PROGRAM BasketToleranceCtrl
VAR
	ARfbStnToleranceCtrl		: ARRAY [0..iStnQty] OF fbToleranceTimeCtrl;

	tArm1ToleranceTimer		: TON;
	tArm1ToleranceTimerEV	: TIME;

	tArm2ToleranceTimer		: TON;
	tArm2ToleranceTimerEV	: TIME;

END_VAR

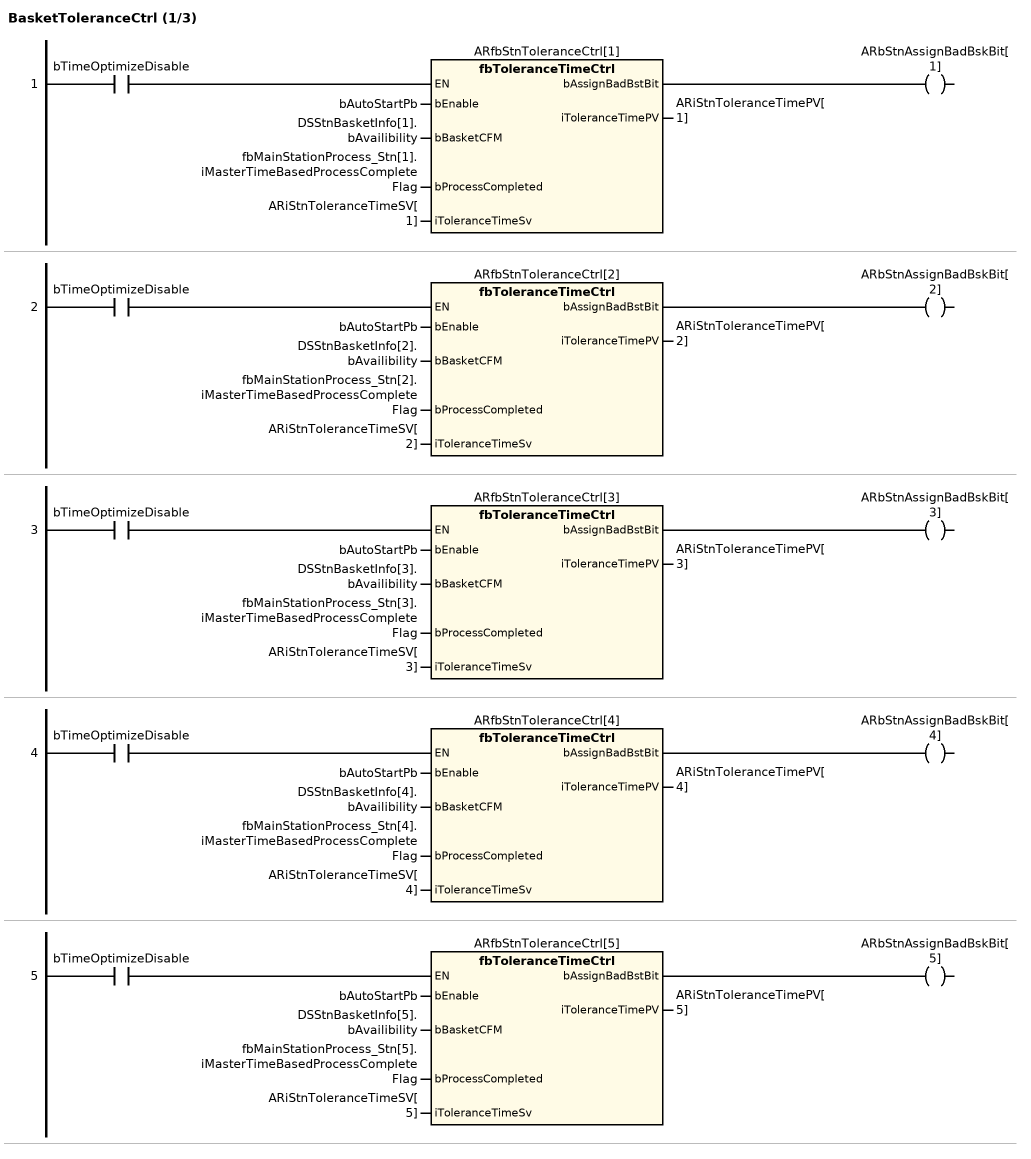
// NETWORK 1
IF bTimeOptimizeDisable THEN
    ARfbStnToleranceCtrl[1](
        bEnable := bAutoStartPb,
        bBasketCFM := DSStnBasketInfo[1].bAvailibility,
        bProcessCompleted := fbMainStationProcess_Stn[1].iMasterTimeBasedProcessCompleteFlag,
        iToleranceTimeSv := ARiStnToleranceTimeSV[1],
        iToleranceTimePV => ARiStnToleranceTimePV[1]); // fbToleranceTimeCtrl
END_IF
ARbStnAssignBadBskBit[1] := ARfbStnToleranceCtrl[1].bAssignBadBstBit;

// NETWORK 2
IF bTimeOptimizeDisable THEN
    ARfbStnToleranceCtrl[2](
        bEnable := bAutoStartPb,
        bBasketCFM := DSStnBasketInfo[2].bAvailibility,
        bProcessCompleted := fbMainStationProcess_Stn[2].iMasterTimeBasedProcessCompleteFlag,
        iToleranceTimeSv := ARiStnToleranceTimeSV[2],
        iToleranceTimePV => ARiStnToleranceTimePV[2]); // fbToleranceTimeCtrl
END_IF
ARbStnAssignBadBskBit[2] := ARfbStnToleranceCtrl[2].bAssignBadBstBit;

// NETWORK 3
IF bTimeOptimizeDisable THEN
    ARfbStnToleranceCtrl[3](
        bEnable := bAutoStartPb,
        bBasketCFM := DSStnBasketInfo[3].bAvailibility,
        bProcessCompleted := fbMainStationProcess_Stn[3].iMasterTimeBasedProcessCompleteFlag,
        iToleranceTimeSv := ARiStnToleranceTimeSV[3],
        iToleranceTimePV => ARiStnToleranceTimePV[3]); // fbToleranceTimeCtrl
END_IF
ARbStnAssignBadBskBit[3] := ARfbStnToleranceCtrl[3].bAssignBadBstBit;

// NETWORK 4
IF bTimeOptimizeDisable THEN
    ARfbStnToleranceCtrl[4](
        bEnable := bAutoStartPb,
        bBasketCFM := DSStnBasketInfo[4].bAvailibility,
        bProcessCompleted := fbMainStationProcess_Stn[4].iMasterTimeBasedProcessCompleteFlag,
        iToleranceTimeSv := ARiStnToleranceTimeSV[4],
        iToleranceTimePV => ARiStnToleranceTimePV[4]); // fbToleranceTimeCtrl
END_IF
ARbStnAssignBadBskBit[4] := ARfbStnToleranceCtrl[4].bAssignBadBstBit;

// NETWORK 5
IF bTimeOptimizeDisable THEN
    ARfbStnToleranceCtrl[5](
        bEnable := bAutoStartPb,
        bBasketCFM := DSStnBasketInfo[5].bAvailibility,
        bProcessCompleted := fbMainStationProcess_Stn[5].iMasterTimeBasedProcessCompleteFlag,
        iToleranceTimeSv := ARiStnToleranceTimeSV[5],
        iToleranceTimePV => ARiStnToleranceTimePV[5]); // fbToleranceTimeCtrl
END_IF
ARbStnAssignBadBskBit[5] := ARfbStnToleranceCtrl[5].bAssignBadBstBit;

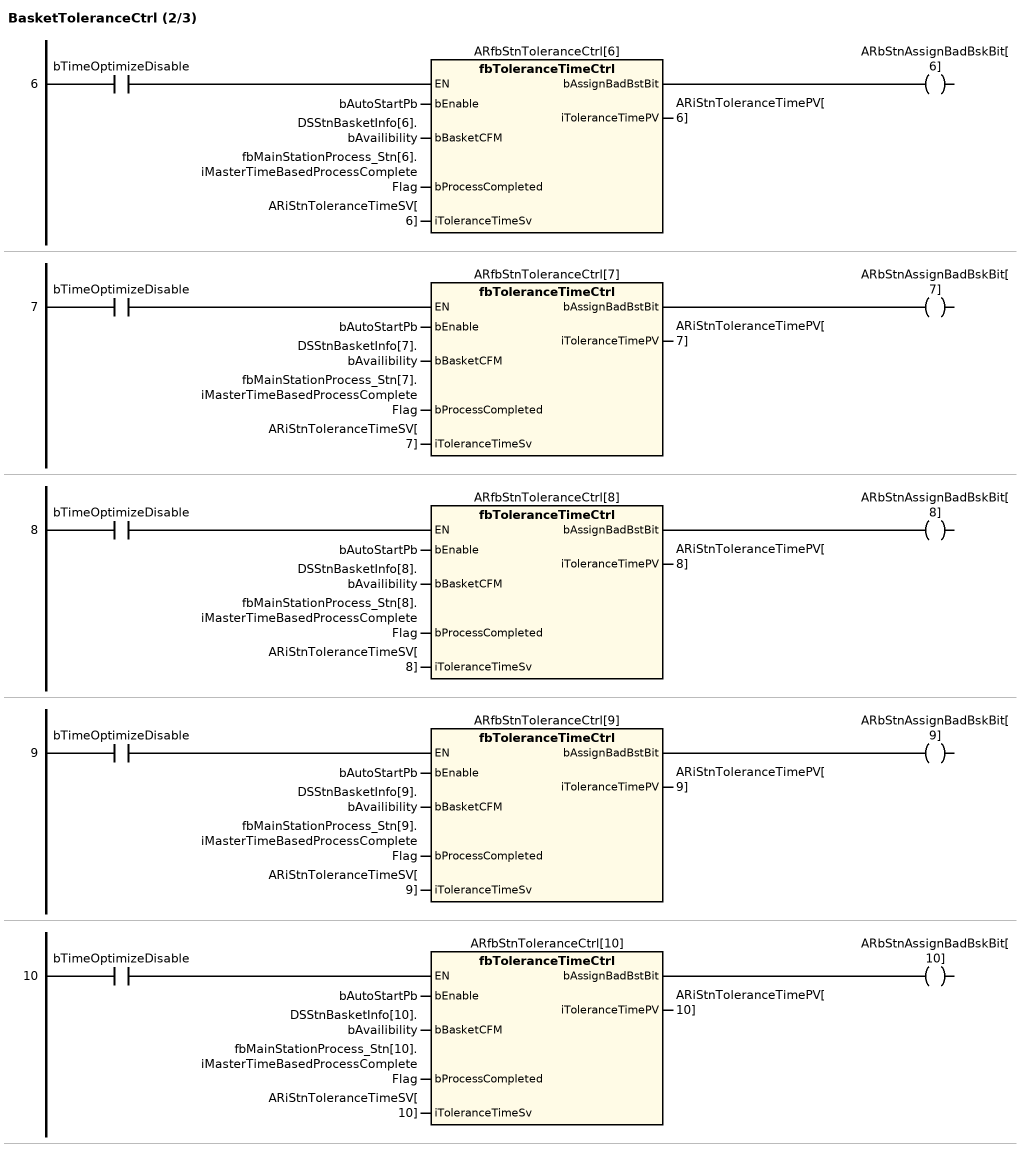
// NETWORK 6
IF bTimeOptimizeDisable THEN
    ARfbStnToleranceCtrl[6](
        bEnable := bAutoStartPb,
        bBasketCFM := DSStnBasketInfo[6].bAvailibility,
        bProcessCompleted := fbMainStationProcess_Stn[6].iMasterTimeBasedProcessCompleteFlag,
        iToleranceTimeSv := ARiStnToleranceTimeSV[6],
        iToleranceTimePV => ARiStnToleranceTimePV[6]); // fbToleranceTimeCtrl
END_IF
ARbStnAssignBadBskBit[6] := ARfbStnToleranceCtrl[6].bAssignBadBstBit;

// NETWORK 7
IF bTimeOptimizeDisable THEN
    ARfbStnToleranceCtrl[7](
        bEnable := bAutoStartPb,
        bBasketCFM := DSStnBasketInfo[7].bAvailibility,
        bProcessCompleted := fbMainStationProcess_Stn[7].iMasterTimeBasedProcessCompleteFlag,
        iToleranceTimeSv := ARiStnToleranceTimeSV[7],
        iToleranceTimePV => ARiStnToleranceTimePV[7]); // fbToleranceTimeCtrl
END_IF
ARbStnAssignBadBskBit[7] := ARfbStnToleranceCtrl[7].bAssignBadBstBit;

// NETWORK 8
IF bTimeOptimizeDisable THEN
    ARfbStnToleranceCtrl[8](
        bEnable := bAutoStartPb,
        bBasketCFM := DSStnBasketInfo[8].bAvailibility,
        bProcessCompleted := fbMainStationProcess_Stn[8].iMasterTimeBasedProcessCompleteFlag,
        iToleranceTimeSv := ARiStnToleranceTimeSV[8],
        iToleranceTimePV => ARiStnToleranceTimePV[8]); // fbToleranceTimeCtrl
END_IF
ARbStnAssignBadBskBit[8] := ARfbStnToleranceCtrl[8].bAssignBadBstBit;

// NETWORK 9
IF bTimeOptimizeDisable THEN
    ARfbStnToleranceCtrl[9](
        bEnable := bAutoStartPb,
        bBasketCFM := DSStnBasketInfo[9].bAvailibility,
        bProcessCompleted := fbMainStationProcess_Stn[9].iMasterTimeBasedProcessCompleteFlag,
        iToleranceTimeSv := ARiStnToleranceTimeSV[9],
        iToleranceTimePV => ARiStnToleranceTimePV[9]); // fbToleranceTimeCtrl
END_IF
ARbStnAssignBadBskBit[9] := ARfbStnToleranceCtrl[9].bAssignBadBstBit;

// NETWORK 10
IF bTimeOptimizeDisable THEN
    ARfbStnToleranceCtrl[10](
        bEnable := bAutoStartPb,
        bBasketCFM := DSStnBasketInfo[10].bAvailibility,
        bProcessCompleted := fbMainStationProcess_Stn[10].iMasterTimeBasedProcessCompleteFlag,
        iToleranceTimeSv := ARiStnToleranceTimeSV[10],
        iToleranceTimePV => ARiStnToleranceTimePV[10]); // fbToleranceTimeCtrl
END_IF
ARbStnAssignBadBskBit[10] := ARfbStnToleranceCtrl[10].bAssignBadBstBit;

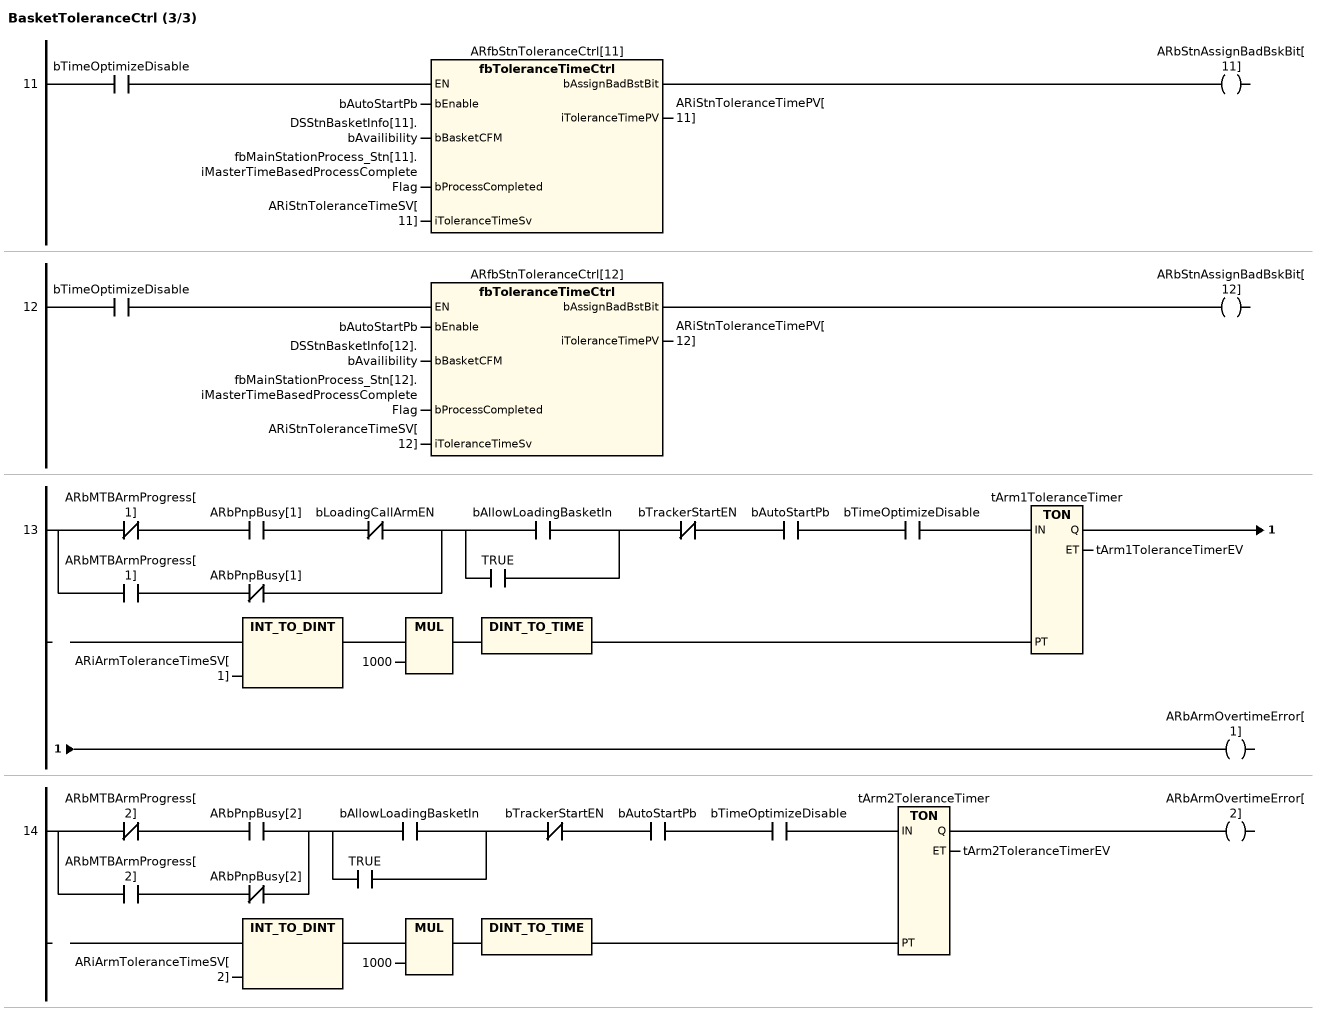
// NETWORK 11
IF bTimeOptimizeDisable THEN
    ARfbStnToleranceCtrl[11](
        bEnable := bAutoStartPb,
        bBasketCFM := DSStnBasketInfo[11].bAvailibility,
        bProcessCompleted := fbMainStationProcess_Stn[11].iMasterTimeBasedProcessCompleteFlag,
        iToleranceTimeSv := ARiStnToleranceTimeSV[11],
        iToleranceTimePV => ARiStnToleranceTimePV[11]); // fbToleranceTimeCtrl
END_IF
ARbStnAssignBadBskBit[11] := ARfbStnToleranceCtrl[11].bAssignBadBstBit;

// NETWORK 12
IF bTimeOptimizeDisable THEN
    ARfbStnToleranceCtrl[12](
        bEnable := bAutoStartPb,
        bBasketCFM := DSStnBasketInfo[12].bAvailibility,
        bProcessCompleted := fbMainStationProcess_Stn[12].iMasterTimeBasedProcessCompleteFlag,
        iToleranceTimeSv := ARiStnToleranceTimeSV[12],
        iToleranceTimePV => ARiStnToleranceTimePV[12]); // fbToleranceTimeCtrl
END_IF
ARbStnAssignBadBskBit[12] := ARfbStnToleranceCtrl[12].bAssignBadBstBit;

// NETWORK 13
tArm1ToleranceTimer(
    IN := ((NOT ARbMTBArmProgress[1] AND ARbPnpBusy[1] AND NOT bLoadingCallArmEN OR ARbMTBArmProgress[1] AND NOT ARbPnpBusy[1]) AND (bAllowLoadingBasketIn OR TRUE)) AND NOT bTrackerStartEN AND bAutoStartPb AND bTimeOptimizeDisable,
    PT := DINT_TO_TIME(INT_TO_DINT(ARiArmToleranceTimeSV[1]) * 1000),
    ET => tArm1ToleranceTimerEV); // TON
ARbArmOvertimeError[1] := tArm1ToleranceTimer.Q;

// NETWORK 14
tArm2ToleranceTimer(
    IN := ((NOT ARbMTBArmProgress[2] AND ARbPnpBusy[2] OR ARbMTBArmProgress[2] AND NOT ARbPnpBusy[2]) AND (bAllowLoadingBasketIn OR TRUE)) AND NOT bTrackerStartEN AND bAutoStartPb AND bTimeOptimizeDisable,
    PT := DINT_TO_TIME(INT_TO_DINT(ARiArmToleranceTimeSV[2]) * 1000),
    ET => tArm2ToleranceTimerEV); // TON
ARbArmOvertimeError[2] := tArm2ToleranceTimer.Q;

END_PROGRAM

(* stored: Version 1.1.0.1, ProductVersion 3.1.4024.12
   POU BasketToleranceCtrl: Id {666660bc-3125-4e33-9555-0639dd6d299a}, SpecialFunc None *)
